// TIA Portal V18 export
// export: Created 2026-06-08T16:04:36.803552Z, ExportSetting WithDefaults, DisplayName Totally Integrated Automation Portal, DisplayVersion V18, DisplayName TIA Portal Openness, DisplayVersion V18, DisplayName TIA Portal Version Control Interface, DisplayVersion V18, DisplayName STEP 7 Professional, DisplayVersion V18, DisplayName STEP 7 Safety, DisplayVersion V18, DisplayName WinCC Professional, DisplayVersion V18
VAR_GLOBAL   // PLC tag table "OUTPUT"
   Q_lamp_Auto AT %Q0.0 : Bool;   // Đèn chế độ auto
   Q_lamp_Manu AT %Q0.1 : Bool;   // Đèn chế độ manu
   Q_BT AT %Q0.2 : Bool;   // Băng tải phân loại
   Q_Xylanh_Cao AT %Q0.3 : Bool;   // Xi lanh đẩy sản phẩm cao
   Q_Xylanh_TB AT %Q0.4 : Bool;   // Xi lanh đẩy sản phẩm trung bình
END_VAR
